{attribute 'qualified_only'}
{attribute 'strict'}
TYPE E_BlackJackVariation :
(
	Idle				:= 0,
	Common_BlackJack 	:= 1,
	FreeBet_BlackJack	:= 2,
	Spanish21			:= 3
	
);
END_TYPE

(* stored: Version 1.1.0.1, ProductVersion 3.1.4024.10
   DUT E_BlackJackVariation: Id {f8fad10b-adf1-4b4e-8cfa-2aaab8b084de} *)
